// TwinCAT 3 PLC project StackerCrane
// ProgramVersion: 3.1.4023.0
// libraries:
//   Tc2_Standard, * (Beckhoff Automation GmbH)
//   Tc2_System, * (Beckhoff Automation GmbH)
//   Tc3_Module, * (Beckhoff Automation GmbH)
// project tree:
//   DUTs/ AdsCom.TcDUT, Outputs.TcDUT, Inputs.TcDUT
//   GVLs/ GVL_ADS.TcGVL, GVL_IO.TcGVL, GVL_Processes.TcGVL
//   / PlcTask.TcTTO
//   POUs/ CraneMovement.TcPOU, Empty.TcPOU, Fill.TcPOU, Home.TcPOU, MAIN.TcPOU, StackerCraneProcess.TcPOU
// real-time tasks:
//   TASK PlcTask: cycle T#10ms, priority 20, ADS port 350

CONFIGURATION StackerCrane
    RESOURCE PLC ON TwinCAT3
        TASK PlcTask(INTERVAL := T#10ms, PRIORITY := 20);
        PROGRAM MAIN WITH PlcTask : MAIN;
    END_RESOURCE
END_CONFIGURATION

// ---- DUTs/AdsCom.TcDUT
TYPE AdsCom :
STRUCT
	iMode : INT := 1;
	iAlgo : INT := 1;
	iRackSlot : INT:=0;
	iTotalPalletsProcessed : INT;
	iPalletsInRack : INT;
	sCurrentOperation : STRING;
	bStart : BOOL;
	bStop : BOOL;
	bHalt : BOOL;
	bResume : BOOL;
	aSlots : ARRAY[1..54] OF BOOL;
END_STRUCT
END_TYPE

// ---- DUTs/Outputs.TcDUT
TYPE Outputs :
STRUCT
	bEntryRollerConveyor: BOOL;
	bExitRollerConveyor: BOOL;
	bEntryLoadingConveyor : BOOL;
	bExitLoadingConveyor : BOOL;
	bEmitPallet : BOOL;
	bSCLift : BOOL;
	bSCLeft : BOOL;
	bSCRight : BOOL;
	iSCPosition : INT;
END_STRUCT
END_TYPE

// ---- DUTs/Inputs.TcDUT
TYPE Inputs :
STRUCT
	bEntrySensor : BOOL;
	bExitSensor : BOOL;
	bSCMovingX : BOOL;
	bSCMovingZ : BOOL;
	bSCLeftLimit : BOOL;
	bSCRightLimit : BOOL;
	bSCMiddlLimit : BOOL;
	
END_STRUCT
END_TYPE

// ---- GVLs/GVL_ADS.TcGVL
VAR_GLOBAL
	stAdsCom : AdsCom;
END_VAR

// ---- GVLs/GVL_IO.TcGVL
VAR_GLOBAL
	{attribute 'OPC.UA.DA' := '1'}
	fioInputs : Inputs;
	
	{attribute 'OPC.UA.DA' := '1'}
	fioOutputs : Outputs;
END_VAR

// ---- GVLs/GVL_Processes.TcGVL
VAR_GLOBAL
	stackerCraneProcess : StackerCraneProcess;
END_VAR

// ---- POUs/MAIN.TcPOU
PROGRAM MAIN
VAR
	
END_VAR

stackerCraneProcess(
	bHalt:=GVL_ADS.stAdsCom.bHalt,
	bResume:=GVL_ADS.stAdsCom.bResume,
	bStart:=GVL_ADS.stAdsCom.bStart,
	bStop:=GVL_ADS.stAdsCom.bStop,
	fioOutputs:=GVL_IO.fioOutputs,
	fioInputs:=GVL_IO.fioInputs,
	iAlgo:=GVL_ADS.stAdsCom.iAlgo,
	iMode:=GVL_ADS.stAdsCom.iMode,
	sCurrentOperation=>GVL_ADS.stAdsCom.sCurrentOperation,
	iPalletsInRack=>GVL_ADS.stAdsCom.iPalletsInRack,
	iTotalPalletsProcessed=>GVL_ADS.stAdsCom.iTotalPalletsProcessed,
	aSlots=>GVL_ADS.stAdsCom.aSlots);

END_PROGRAM

// ---- POUs/StackerCraneProcess.TcPOU
FUNCTION_BLOCK StackerCraneProcess
VAR_IN_OUT
	bStart : BOOL;
	bHalt : BOOL;
	bResume : BOOL;
	bStop : BOOL;
	fioOutputs : OUTPUTS;
END_VAR
VAR_INPUT
	fioInputs : INPUTS;
	iAlgo: INT;
	iMode: INT;
END_VAR
VAR_OUTPUT
	sCurrentOperation : STRING;
	iTotalPalletsProcessed : INT;
	iPalletsInRack : INT;
	aSlots : ARRAY[1..54] OF BOOL;

END_VAR
VAR
	iStep : INT;
	startTrig : R_TRIG;
	stopTrig : R_TRIG;
	resumeTrig : R_TRIG;
	haltTrig : R_TRIG;
	iHaltStep : INT;
	mAlgo : INT;
	mMode : INT;
	i : INT;
	iChosenSlot : INT;
	fill : Fill;
	empty : Empty;
	iCounter :INT;
	exitTimer : TON;
END_VAR

VAR CONSTANT
	AVAILABLE_SLOTS: INT := 54;
END_VAR

startTrig(CLK:=bStart);
stopTrig(CLK:=bStop);
resumeTrig(CLK:=bResume);
haltTrig(CLK:=bHalt);
exitTimer(PT:=T#5S);

fill(
	fioOutputs:=fioOutputs,
	iPalletsInRack:=iPalletsInRack,
	sCurrentOperation:=sCurrentOperation,
	aSlots:=aSlots,
	fioInputs:=fioInputs);
	
empty(
	fioOutputs:=fioOutputs,
	iPalletsInRack:=iPalletsInRack,
	sCurrentOperation:=sCurrentOperation,
	aSlots:=aSlots,
	fioInputs:=fioInputs);	
	
IF startTrig.Q 
	AND iStep = 0
	THEN
	resetInputs();
	mAlgo := iAlgo;
	mMode := iMode;
	iStep := 10;
END_IF

IF resumeTrig.Q 
	AND iStep  = 1000
	THEN
	resetInputs();
	iStep := iHaltStep;	
END_IF

IF haltTrig.Q
	THEN
	resetInputs();
	iHaltStep := iStep;
	iStep := 1000;	
END_IF

IF stopTrig.Q
	THEN
	resetInputs();
	exitTimer.IN := FALSE;
	iStep :=  2000;
END_IF

CASE iStep OF
	0:
	 	sCurrentOperation := 'Idle';
		resetInputs();

	10: 
		IF mMode = 1 // Fill
			AND iPalletsInRack < 54
			THEN
			iTotalPalletsProcessed := iTotalPalletsProcessed + 1;
			// Emit Pallet
			fioOutputs.bEmitPallet := TRUE;
			// Start Entry Conveyors
			fioOutputs.bEntryRollerConveyor := TRUE;
			fioOutputs.bEntryLoadingConveyor := TRUE;
			sCurrentOperation := 'Entry Conveyor started';
			iStep := 20;
		ELSIF mMode = 2
			AND iPalletsInRack > 0 // empty
			THEN
			iStep := 60;
			
		ELSE // Not mplemented yet
			iStep := 0;
		END_IF
		
	// ------------------------------------------------------------------------ Fill operation --------------------------------------------------------
	20: // Check Pallet in Loading Conveyor
		IF fioInputs.bEntrySensor
			THEN
			// Stop emitting and stop conveyors
			fioOutputs.bEntryRollerConveyor := FALSE;
			fioOutputs.bEntryLoadingConveyor := FALSE;
			fioOutputs.bEmitPallet := FALSE;	
			iStep := 30;	
		END_IF
		
	30: // Check if space available in rack
		IF iPalletsInRack < AVAILABLE_SLOTS
			THEN
			iStep := 40;
		ELSE
			// Halt operations
			iStep := 1000;
		END_IF
		
	40: // Check algo for fill operation
	
		IF mAlgo = 1 // Sequential
			THEN
			sCurrentOperation := 'Filling sequentially';
			FOR i := 1 TO 54 DO
				IF aSlots[i] = FALSE
					THEN
					iChosenSlot := i;
					EXIT;
				END_IF
			END_FOR
			iStep := 50;
		ELSE
			// Halt operations
			iStep := 1000;
		END_IF
		
	50:
		fill.bStart := TRUE;
		fill.iSlotPosition := iChosenSlot;
		IF fill.bDone THEN
			fill.bStart := FALSE;
			iStep := 0;
		END_IF
		
		
	// ------------------------------------------------------------------------ Empty operation --------------------------------------------------------
	60: //Check algo for empty operation
	
		IF mAlgo = 1 // Sequential
			THEN
			sCurrentOperation := 'Emptying sequentially';
			iCounter := 54;
			WHILE iCounter<>0 DO
				IF aSlots[iCounter] 
					THEN
					iChosenSlot := iCounter;
					EXIT;
				END_IF
    			iCounter := iCounter-1;
			END_WHILE
			
			iStep := 70;
		ELSE
			// Halt operations
			iStep := 1000;
		END_IF
		
	70:
		empty.bStart := TRUE;
		empty.iSlotPosition := iChosenSlot;
		IF empty.bDone THEN
			empty.bStart := FALSE;
			iStep := 80;
		END_IF
		
	80:
		fioOutputs.bExitLoadingConveyor := TRUE;
		fioOutputs.bExitRollerConveyor := TRUE;
		IF fioInputs.bExitSensor
			THEN
			iStep := 90;
		END_IF
		
	90:
		exitTimer.IN := TRUE;
		IF exitTimer.Q
			THEN
			exitTimer.IN := FALSE;
			fioOutputs.bExitLoadingConveyor := FALSE;
			fioOutputs.bExitRollerConveyor := FALSE;
			iStep:=0;
		END_IF
END_CASE

METHOD PRIVATE resetInputs : BOOL
VAR_INPUT
END_VAR
bStart := FALSE;
bHalt := FALSE;
bResume := FALSE;
bStop := FALSE;
END_METHOD

END_FUNCTION_BLOCK

// ---- POUs/Fill.TcPOU
FUNCTION_BLOCK Fill EXTENDS CraneMovement
VAR_INPUT
END_VAR
VAR_OUTPUT
END_VAR
VAR
END_VAR

SUPER^(
	iPalletsInRack:=iPalletsInRack,
	aSlots:=aSlots,
	fioOutputs:=fioOutputs,
	sCurrentOperation:=sCurrentOperation);
	
IF bStart 
	AND iStep = 0
	AND iPalletsInRack < 54
	THEN
	iStep := 10;
	bBusy := TRUE;
ELSIF NOT bStart
	THEN
	bDone := FALSE;
	bBusy := FALSE;
	iStep := 0;
END_IF


CASE iStep OF
	
	10: // Start loading pallet on the stacker crane 
	(* 
		Entering critical process section:
		If the process is stopped here, particular care is needed to recover
		and make sure that the pallet is either stored in the chosen slot or 
		removed from the line
	*)
		fioOutputs.bSCRight := TRUE;
		IF fioInputs.bSCRightLimit 
			THEN
			iStep := 20;
		END_IF
		
	20: // Lift the stacker crane
	
		fioOutputs.bSCLift := TRUE;
		liftTimer.IN := TRUE;
		
		IF liftTimer.Q
			THEN
			liftTimer.IN := FALSE;
			iStep := 30;
		END_IF
		
	30: // Stacker crane in middle position
	
		fioOutputs.bSCRight := FALSE;
		IF fioInputs.bSCMiddlLimit
			THEN
			istep := 40;
		END_IF
		
	40: // Lower stacker crane
		
		fioOutputs.bSCLift := FALSE;
		liftTimer.IN := TRUE;
		
		IF liftTimer.Q
			THEN
			liftTimer.IN := FALSE;
			iStep := 50;
		END_IF
	
	50: // Go to required position
	
		sCurrentOperation := Concat('Going to slot position ', INT_TO_STRING(iSlotPosition));
		fioOutputs.iSCPosition := iSlotPosition;
		motionTimer.IN := TRUE;
		
		IF NOT fioInputs.bSCMovingX
			 AND NOT fioInputs.bSCMovingZ
			 AND motionTimer.Q
			 THEN
			 
			 motionTimer.IN := FALSE;
			 iStep := 60; 
		END_IF
		
	60: // Lift 
	
		fioOutputs.bSCLift := TRUE;
		liftTimer.IN := TRUE;
		
		IF liftTimer.Q
			THEN
			liftTimer.IN := FALSE;
			iStep := 70;
		END_IF
	
	70: // Unload into the rack
		sCurrentOperation := 'Unloading';
		fioOutputs.bSCLeft := TRUE;
		IF fioInputs.bSCLeftLimit
			THEN
			istep := 80;
		END_IF
	
	80: // Lower the crane
	
		fioOutputs.bSCLift := FALSE;
		liftTimer.IN := TRUE;
		
		IF liftTimer.Q
			THEN
			aSlots[iSlotPosition] := TRUE;
			iPalletsInRack:=iPalletsInRack+1;
			liftTimer.IN := FALSE;
			iStep := 90;
		END_IF
	
	90: // Return to the middle position
		sCurrentOperation := 'Return to initial position';
		fioOutputs.bSCLeft := FALSE;
		IF fioInputs.bSCMiddlLimit
			THEN
			istep := 100;
		END_IF	
		
	100: // Return to the load position
	
		fioOutputs.iSCPosition := 55;
		motionTimer.IN := TRUE;
		
		IF NOT fioInputs.bSCMovingX
			 AND NOT fioInputs.bSCMovingZ
			 AND motionTimer.Q
			 THEN
			 motionTimer.IN := FALSE;
			 bDone := TRUE;
			 bBusy := FALSE;
			 iStep := 110; 
		END_IF
	
END_CASE

END_FUNCTION_BLOCK

// ---- POUs/CraneMovement.TcPOU
FUNCTION_BLOCK CraneMovement
VAR_IN_OUT
	fioOutputs : OUTPUTS;
	iPalletsInRack : INT;
	aSlots : ARRAY[1..54] OF BOOL;
	sCurrentOperation : STRING;
END_VAR

VAR_INPUT
	bStart : BOOL;
	fioInputs : INPUTS;
	iSlotPosition : INT;
END_VAR

VAR_OUTPUT
	bBusy : BOOL;
	bDone : BOOL;
END_VAR

VAR
	iStep : INT;
	startTrig : R_TRIG;
	stopTrig : R_TRIG;
	resumeTrig : R_TRIG;
	haltTrig : R_TRIG;
	iHaltStep : INT;
	mAlgo : INT;
	mMode : INT;
	i : INT;
	iChosenSlot : INT;
	liftTimer : TON;
	motionTimer : TON;
END_VAR

liftTimer(PT:=T#2S); 
motionTimer(PT:=T#1S);

END_FUNCTION_BLOCK

// ---- POUs/Empty.TcPOU
FUNCTION_BLOCK Empty EXTENDS CraneMovement
VAR_INPUT
END_VAR
VAR_OUTPUT
END_VAR
VAR
END_VAR

SUPER^(
	iPalletsInRack:=iPalletsInRack,
	aSlots:=aSlots,
	fioOutputs:=fioOutputs,
	sCurrentOperation:=sCurrentOperation);
	
IF bStart 
	AND iStep = 0
	and iPalletsInRack > 0
	THEN
	iStep := 10;
	bBusy := TRUE;
ELSIF NOT bStart
	THEN
	bDone := FALSE;
	bBusy := FALSE;
	iStep := 0;
END_IF


CASE iStep OF
	

	10: // Go to required position
	
		sCurrentOperation := Concat('Going to slot position ', INT_TO_STRING(iSlotPosition));
		fioOutputs.iSCPosition := iSlotPosition;
		motionTimer.IN := TRUE;
		
		IF NOT fioInputs.bSCMovingX
			 AND NOT fioInputs.bSCMovingZ
			 AND motionTimer.Q
			 THEN
			 
			 motionTimer.IN := FALSE;
			 iStep := 20; 
		END_IF
		
	20: // load the pallet on the stacker crane
		sCurrentOperation := 'Loading';
		fioOutputs.bSCLeft := TRUE;
		IF fioInputs.bSCLeftLimit
			THEN
			istep := 30;
		END_IF
		
	30: // Lift 
	
		fioOutputs.bSCLift := TRUE;
		liftTimer.IN := TRUE;
		
		IF liftTimer.Q
			THEN
			liftTimer.IN := FALSE;
			iStep := 40;
		END_IF
		
	40: // Stacker crane in middle position
	
		fioOutputs.bSCLeft := FALSE;
		IF fioInputs.bSCMiddlLimit
			THEN
			istep := 50;
		END_IF	
		
	50: // Lower the crane
	
		fioOutputs.bSCLift := FALSE;
		liftTimer.IN := TRUE;
		
		IF liftTimer.Q
			THEN
			aSlots[iSlotPosition] := FALSE;
			iPalletsInRack:=iPalletsInRack-1;
			liftTimer.IN := FALSE;
			iStep := 60;
		END_IF
	
		
	60: // Return to the load position
		sCurrentOperation := 'Return to initial position';

		fioOutputs.iSCPosition := 55;
		motionTimer.IN := TRUE;
		
		IF NOT fioInputs.bSCMovingX
			 AND NOT fioInputs.bSCMovingZ
			 AND motionTimer.Q
			 THEN
			 motionTimer.IN := FALSE;
			
			 iStep := 70; 
		END_IF
		
	70: // Lift the stacker crane
	
		fioOutputs.bSCLift := TRUE;
		liftTimer.IN := TRUE;
		
		IF liftTimer.Q
			THEN
			liftTimer.IN := FALSE;
			iStep := 80;
		END_IF
		
	80: // Start loading pallet on the stacker crane 
	
		fioOutputs.bSCLeft := TRUE;
		IF fioInputs.bSCLeftLimit 
			THEN
			iStep := 90;
		END_IF	
		
	90: // Lower stacker crane
		
		fioOutputs.bSCLift := FALSE;
		liftTimer.IN := TRUE;
		
		IF liftTimer.Q
			THEN
			liftTimer.IN := FALSE;
			iStep := 100;
		END_IF	
		
	100: // Return to the middle position
		fioOutputs.bSCLeft := FALSE;
		IF fioInputs.bSCMiddlLimit
			THEN
			bDone := TRUE;
			bBusy := FALSE;
			istep := 110;
		END_IF		

	
	
END_CASE

END_FUNCTION_BLOCK

// ---- POUs/Home.TcPOU
FUNCTION_BLOCK Home extends CraneMovement
VAR_INPUT
END_VAR
VAR_OUTPUT
END_VAR
VAR
END_VAR

END_FUNCTION_BLOCK
